{attribute 'qualified_only'}
{attribute 'strict'}
{attribute 'to_string'}
TYPE E_MOVER_SELECTOR :
(
	SELECT_MOVER_INDEX,
  SELECT_MOVER_AXIS_ID
);
END_TYPE

(* stored: Version 1.1.0.1, ProductVersion 3.1.4026.18
   DUT E_MOVER_SELECTOR: Id {6c705f32-52ee-42ab-99cd-e3c6839ae66e} *)
